INTERFACE I_EpicsMotionParamsStatus

METHOD MotionParamsAndStatus
VAR_INPUT
	PowerEnabled : BOOL;
	PowerIsEnabled : BOOL;
	Execute : BOOL;
	LimHome : BOOL;
	MoveBackwardEnabled : BOOL;
	MoveForwardEnabled : BOOL;
	MeasuredPositionDiff : LREAL;
	MeasuredPosition : LREAL;
	MeasuredVelocity : LREAL;
	PowerOverride : LREAL;
	Busy : BOOL;
	HomeDone : BOOL;
END_VAR
END_METHOD

END_INTERFACE

(* stored: Version 1.1.0.1
   Itf I_EpicsMotionParamsStatus: Id {02fc6aae-4594-4c34-9af1-4c410ddc4a58}
   Method MotionParamsAndStatus: Id {aab41c89-baf0-4400-9d56-890b81c35521} *)
